{attribute 'qualified_only'}
{attribute 'strict'}
TYPE E_Gen24_Error :
(
	eNoError := 0,
	eModbusTCPError := 1,
	eGen24Error := 2,
	eGen24TooBigValueReceived := 3
);
END_TYPE

(* stored: Version 1.1.0.1, ProductVersion 3.1.4024.6
   DUT E_Gen24_Error: Id {67fb49dd-ff1c-4da9-9445-3fca295cadb9} *)
